PROGRAM PRG_TEST
VAR
	HeatingCurve_Test : FC_HeatingCurve_Test;							 
END_VAR

TcUnit.RUN();

END_PROGRAM

(* stored: Version 1.1.0.1, ProductVersion 3.1.4024.6
   POU PRG_TEST: Id {0cbfb4b1-94b7-40de-9fdc-5d0f41511cae}, SpecialFunc None *)
